FUNCTION_BLOCK DFB_FacilityAlarmBool
VAR_INPUT
	Sec_P					: BOOL; // Second pulse
	TbotNo					: INT; // 1: Tbot left, 2: Tbot right
	InputWarning			: BOOL;
	InputAlarm				: BOOL;
	WarningTimer			: UDINT;
	AlarmTimer				: UDINT;
	AbortTimer				: UDINT;
	LogName					: STRING;
	ModuleID				: E_ModuleID;
	EventName				: E_EventName;
END_VAR

VAR_OUTPUT
	OutputWarning			: BOOL;
	OutputAlarm				: BOOL;
	OutputAbort				: BOOL;
END_VAR

VAR
	_State_Changed			: BOOL;
	
	_State					: INT;
	_Last_State				: INT;
	_TLast_State			: INT;
	
	_State_Timer			: UDINT;
	
	_EmptyEvent				: ST_Event;
	
	_TON_Warning			: TON;
	_TON_Alarm				: TON;				
END_VAR

///////////////////////////////////////////////////////////////////////////////////////////////////////////////////////////////////////////////////////////////////////////////
//	State timer
///////////////////////////////////////////////////////////////////////////////////////////////////////////////////////////////////////////////////////////////////////////////

_State_Changed									:= _State <> _TLast_State;
_TLast_State									:= _State;

IF _State_Changed THEN
	_State_Timer								:= 0;
	Logging.fbDebugLog.M_nLogger(iLogLevel:= iLogVerbosity, sSource:= ' SEQ Log ', 
		sMessage								:= CONCAT(CONCAT(LogName, 'current state['),
														 CONCAT(INT_TO_STRING(_State), ']'))); 
	
ELSE
	IF Sec_P THEN
		_State_Timer							:= _State_Timer + 1;
	END_IF
END_IF

///////////////////////////////////////////////////////////////////////////////////////////////////////////////////////////////////////////////////////////////////////////////
//	State case
///////////////////////////////////////////////////////////////////////////////////////////////////////////////////////////////////////////////////////////////////////////////

CASE _State OF
	0: (*Idle*)
	
		(*Action*)
		OutputWarning							:= FALSE;
		OutputAlarm								:= FALSE;
		OutputAbort								:= FALSE;
		_TON_Warning(IN:= FALSE, PT:= UDINT_TO_TIME(WarningTimer * 1000));
		
		(*Transition*)
		IF InputAlarm THEN
			_TON_Warning(IN:= TRUE, PT:= UDINT_TO_TIME(WarningTimer * 1000));
			_State								:= 21; // Alarm - Delay
		ELSIF InputWarning THEN
			_TON_Warning(IN:= TRUE, PT:= UDINT_TO_TIME(WarningTimer * 1000));
			_State								:= 11; // Warning - Delay
		END_IF
		
	11: (*Warning - Delay*)
		_Last_State								:= 11;
		
		(*Action*)
		OutputWarning							:= FALSE;
		OutputAlarm								:= FALSE;
		OutputAbort								:= FALSE;
		_TON_Warning(IN:= TRUE, PT:= UDINT_TO_TIME(WarningTimer * 1000));
		
		(*Transition*)
		IF (NOT InputWarning) THEN
			_State								:= 0; // Idle
		ELSIF InputAlarm THEN
			_State								:= 21; // Alarm - Delay
		ELSIF _State_Timer >= WarningTimer THEN
			_State								:= 22; // Warning - Send Event
		END_IF
	
	21: (*Alarm - Delay*)
		_Last_State								:= 21;
		
		(*Action*)
		OutputWarning							:= FALSE;
		OutputAlarm								:= FALSE;
		OutputAbort								:= FALSE;
		
		(*Transition*)
		IF (NOT InputAlarm) THEN
			IF InputWarning THEN
				_State							:= 11; // Warning - Delay
			ELSE
				_State							:= 0; // Idle
			END_IF
		ELSIF _State_Timer >= AlarmTimer THEN
			_State								:= 24; // Alarm - Send Event
		END_IF
	
	22:	(*Warning - Send Event*)
		_Last_State								:= 22;
		
		(*Action*)
		OutputWarning							:= TRUE;
		OutputAlarm								:= FALSE;
		OutputAbort								:= FALSE;
		
		// Event - AbortInProgress
		CmdAndEventProcess.fbCmdAndEventUpdate.M_AddEvent(
			sLogName							:= LogName, 
			eEventName							:= EventName, 
			eModuleID							:= ModuleID, 
			iParam								:= _EmptyEvent.iParam,
			sParam								:= _EmptyEvent.sParam, 
			bParam								:= _EmptyEvent.bParam, 
			dParam								:= _EmptyEvent.dParam,
			sFailReason							:= '');
		
		(*Transition*)
		_State									:= 25; // Warning - Check abort time
		
	24: (*Alarm - Send Event*)
		_Last_State								:= 24;
		
		(*Action*)
		OutputWarning							:= FALSE;
		OutputAlarm								:= TRUE;
		OutputAbort								:= FALSE;
		
		// Event - AbortInProgress
		CmdAndEventProcess.fbCmdAndEventUpdate.M_AddEvent(
			sLogName							:= LogName, 
			eEventName							:= EventName, 
			eModuleID							:= ModuleID, 
			iParam								:= _EmptyEvent.iParam,
			sParam								:= _EmptyEvent.sParam, 
			bParam								:= _EmptyEvent.bParam, 
			dParam								:= _EmptyEvent.dParam,
			sFailReason							:= '');
		
		(*Transition*)
		_State									:= 26; // Alarm - Check abort time
		
	25: (*Warning - Check abort time*)
		_Last_State								:= 25;
		
		(*Action*)
		OutputWarning							:= TRUE;
		OutputAlarm								:= FALSE;
		OutputAbort								:= FALSE;
		
		(*Transition*)
		IF _State_Timer >= AbortTimer THEN
			_State								:= 40; // Abort - Warning
		END_IF
		
	26: (*Alarm - Check abort time*)
		_Last_State								:= 26;
		
		(*Action*)
		OutputWarning							:= FALSE;
		OutputAlarm								:= TRUE;
		OutputAbort								:= FALSE;
		
		(*Transition*)
		IF _State_Timer >= AbortTimer THEN
			_State								:= 41; // Abort - Alarm
		END_IF
		
	40: (*Abort - Warning*)
		_Last_State								:= 40;
		
		(*Action*)
		OutputWarning							:= TRUE;
		OutputAlarm								:= FALSE;
		OutputAbort								:= TRUE;
		
		(*Transition*)
		IF (NOT InputWarning) THEN
			_State								:= 0; // Idle
		END_IF
		
	41: (*Abort - Alarm*)
		_Last_State								:= 41;
		
		(*Action*)
		OutputWarning							:= FALSE;
		OutputAlarm								:= TRUE;
		OutputAbort								:= TRUE;
		
		(*Transition*)
		IF (NOT InputWarning) THEN
			_State								:= 0; // Idle
		END_IF
END_CASE

END_FUNCTION_BLOCK

(* stored: Version 1.1.0.1, ProductVersion 3.1.4022.18
   POU DFB_FacilityAlarmBool: Id {20e65b03-5745-4832-829b-b3227b33dae5}, SpecialFunc None *)
